(*
	Link component with additional interface:
	Control BYTE: From TwinCAT >>> To Unity	(Default)
	Status BYTE: FROM Unity >>> TO TwinCAT	(Default)
	ControlData WORD: From TwinCAT >>> To Unity		
	StatusData WORD: FROM Unity >>> TO TwinCAT		
*)
FUNCTION_BLOCK FB_LinkDataWord EXTENDS FB_LinkDevice
VAR	
	{attribute 'simulation_interface'}
	ControlData		AT %Q* : WORD;
	{attribute 'simulation_interface'}
	StatusData		AT %I* : WORD;	
END_VAR

SUPER^();

METHOD INTERNAL GetLinkControlData : WORD
GetLinkControlData := ControlData;
END_METHOD

METHOD INTERNAL SetLinkStatusData : BOOL
VAR_INPUT
	nStatusData : WORD;
END_VAR
StatusData := nStatusData;
END_METHOD

END_FUNCTION_BLOCK

(* stored: Version 1.1.0.1, ProductVersion 3.1.4024.12
   POU FB_LinkDataWord: Id {1027de07-48a8-0ab0-0b84-d0924d9dc9a0}, SpecialFunc None
   Method GetLinkControlData: Id {ea5e0deb-046e-0376-2f82-211873fa08f2}
   Method SetLinkStatusData: Id {218fde2d-3ea4-09b6-140f-7d7b34287882} *)
